FUNCTION_BLOCK ToNcErrorCode_Tests EXTENDS FB_TestSuite

ConversionOfValidErrorCode();
ConversionOfInvalidErrorCode();

METHOD ConversionOfInvalidErrorCode
TcUnit.TEST('ConversionOfInvalidErrorCode');

AssertEquals_DINT(
    Expected:=NcErrorCodes.ERR_UNKNOWN,
    Actual:=ToNcErrorCode(1234567),
    Message:='Error conversion not correct.'
);

TcUnit.TEST_FINISHED();
END_METHOD

METHOD ConversionOfValidErrorCode
TcUnit.TEST('ConversionOfValidErrorCode');

AssertEquals_UDINT(
    Expected:=NcErrorCodes.CONTROLLER_ERROR_DRIVE_ADDRESS,
    Actual:=ToNcErrorCode(17730),
    Message:='Error conversion not correct.'
);

TcUnit.TEST_FINISHED();
END_METHOD

END_FUNCTION_BLOCK

(* stored: Version 1.1.0.1
   POU ToNcErrorCode_Tests: Id {eeee2df2-70e3-0b22-0bc5-56743421a8c2}, SpecialFunc None
   Method ConversionOfInvalidErrorCode: Id {3e4f1ab9-0c8e-0978-369b-6d4bc925d2ff}
   Method ConversionOfValidErrorCode: Id {7468ef5f-d38a-04ed-37df-1008d5c474e3} *)
